// TIA Portal V19 export
FUNCTION_BLOCK "MatLub_FB"   // FB104, LAD
TITLE = MATERIAL LUBRICATION
// stored: MemoryReserve 100, SetENOAutomatically false
   VAR_INPUT
      AreaInterface : "AreaInterface";
      DSI : "udt_DeviceSafetyInterface";
      DataIn : Struct
         Pb_Stop : Bool;
         Pb_Start : Bool;
         SensorLevel : Bool;
      END_STRUCT;
      CoordinationIn : Struct
         MaterialMoving : Bool;
      END_STRUCT;
      Config : Struct
         EnableWngSystemOff : Bool;
         LowTankLevelDly : Time;
      END_STRUCT;
   END_VAR
   VAR_OUTPUT
      MachineInterface : "MachineInterface";
      DataOut : Struct
         SolenoidValve : Bool;
         Lamp : Bool;
      END_STRUCT;
      CoordinationOut : Struct
         IsRunning : Bool;
      END_STRUCT;
   END_VAR
   VAR_IN_OUT
      Parameter : Struct
         SystemOnOff : Bool;
         DelayOff : Time;
      END_STRUCT;
   END_VAR
   VAR
      Sts : Struct
         AlarmsPresence : Bool;
         WarningsPresence : Bool;
         IsStandstill : Bool;
         RunReq : Bool;
         GenCondition { ExternalAccessible := 'False'; ExternalVisible := 'False'; ExternalWritable := 'False'} : Bool;
      END_STRUCT;
      Ctrl : Struct
         RstAlarms : Bool;
         StopDueDoorOpeningRequest : Bool;
         StopSafeStandstill : Bool;
         SafeMotion : Bool;
         StopInPhase : Bool;
         StopProgrammed : Bool;
         StopAborting : Bool;
         ManStart : Bool;
         AutStart : Bool;
      END_STRUCT;
      Alr : Struct
         LowTankLevel : Bool;
      END_STRUCT;
      Wng : Struct
         NoAutReady : Bool;
         SystemOff : Bool;
      END_STRUCT;
      TON_DelayBlowerStop : IEC_TIMER;
      TON_LowTankLevel : IEC_TIMER;
      AckRstAlarms : Bool;
      PbStart_PEAux : Bool;
   END_VAR
   VAR_TEMP   // added for the SCL form of the ladder/FBD networks
      _w1 : Bool;
   END_VAR
BEGIN

REGION Network 1 (SCL): Reset alarms command
   #Ctrl.RstAlarms := #AreaInterface.RstAlarms AND NOT #AckRstAlarms; 
   #AckRstAlarms := #AreaInterface.RstAlarms;

   IF    #Ctrl.RstAlarms THEN
       #Wng.NoAutReady := FALSE;
       #Alr.LowTankLevel := FALSE;
     END_IF;
END_REGION

REGION Network 2: Warning Pump / Blower off
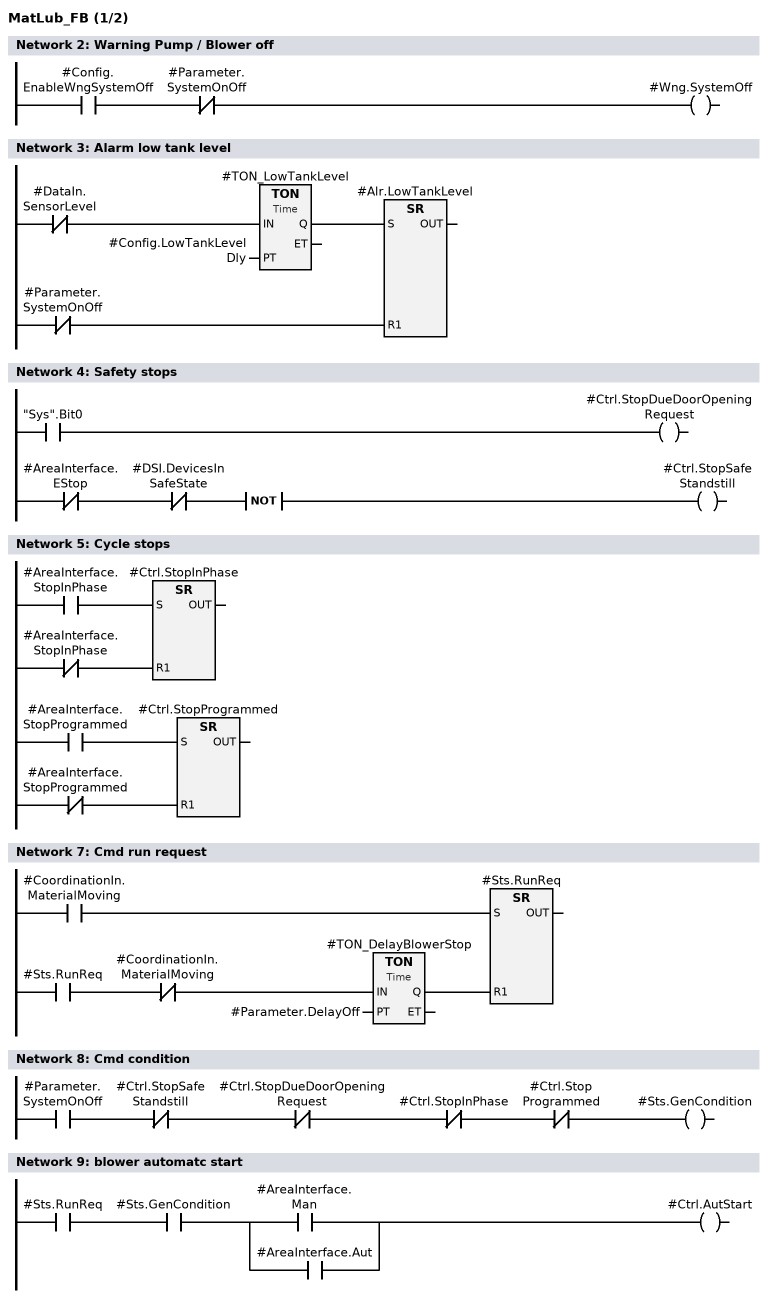
   RUNG wire#powerrail
      Contact( #Config.EnableWngSystemOff )
      I_Contact( #Parameter.SystemOnOff )
      Coil( #Wng.SystemOff )
   END_RUNG
   // the same network as SCL:
   #Wng.SystemOff := #Config.EnableWngSystemOff AND NOT #Parameter.SystemOnOff;
END_REGION

REGION Network 3: Alarm low tank level
   RUNG wire#powerrail
      I_Contact( #DataIn.SensorLevel )
      { S7_Templates := "time_type := Time" } #TON_LowTankLevel.TON(pt := #Config.LowTankLevelDly, et =>)
      S_SR(operand := #Alr.LowTankLevel, r1 := wire#w1)
   END_RUNG
   RUNG wire#powerrail
      I_Contact( #Parameter.SystemOnOff )
   END_RUNG wire#w1
   // the same network as SCL:
   #TON_LowTankLevel.TON(IN := NOT #DataIn.SensorLevel, PT := #Config.LowTankLevelDly);
   IF #TON_LowTankLevel.Q THEN
       #Alr.LowTankLevel := TRUE;   // SR flip-flop
   END_IF;
   IF NOT #Parameter.SystemOnOff THEN #Alr.LowTankLevel := FALSE; END_IF;
END_REGION

REGION Network 4: Safety stops
   RUNG wire#powerrail
      Contact( "Sys".Bit0 )
      Coil( #Ctrl.StopDueDoorOpeningRequest )
   END_RUNG
   RUNG wire#powerrail
      I_Contact( #AreaInterface.EStop )
      I_Contact( #DSI.DevicesInSafeState )
      Not()
      Coil( #Ctrl.StopSafeStandstill )
   END_RUNG
   // the same network as SCL:
   #Ctrl.StopDueDoorOpeningRequest := "Sys".Bit0;
   #Ctrl.StopSafeStandstill := NOT (NOT #AreaInterface.EStop AND NOT #DSI.DevicesInSafeState);
END_REGION

REGION Network 5: Cycle stops
   RUNG wire#powerrail
      Contact( #AreaInterface.StopInPhase )
      S_SR(operand := #Ctrl.StopInPhase, r1 := wire#w1)
   END_RUNG
   RUNG wire#powerrail
      I_Contact( #AreaInterface.StopInPhase )
   END_RUNG wire#w1
   RUNG wire#powerrail
      Contact( #AreaInterface.StopProgrammed )
      S_SR(operand := #Ctrl.StopProgrammed, r1 := wire#w2)
   END_RUNG
   RUNG wire#powerrail
      I_Contact( #AreaInterface.StopProgrammed )
   END_RUNG wire#w2
   // the same network as SCL:
   IF #AreaInterface.StopInPhase THEN
       #Ctrl.StopInPhase := TRUE;   // SR flip-flop
   END_IF;
   IF NOT #AreaInterface.StopInPhase THEN #Ctrl.StopInPhase := FALSE; END_IF;
   IF #AreaInterface.StopProgrammed THEN
       #Ctrl.StopProgrammed := TRUE;   // SR flip-flop
   END_IF;
   IF NOT #AreaInterface.StopProgrammed THEN #Ctrl.StopProgrammed := FALSE; END_IF;
END_REGION

REGION Network 6: <<< BLOWER >>> / <<< COMAMND >>>
END_REGION

REGION Network 7: Cmd run request
   RUNG wire#powerrail
      Contact( #CoordinationIn.MaterialMoving )
      S_SR(operand := #Sts.RunReq, r1 := wire#w1)
   END_RUNG
   RUNG wire#powerrail
      Contact( #Sts.RunReq )
      I_Contact( #CoordinationIn.MaterialMoving )
      { S7_Templates := "time_type := Time" } #TON_DelayBlowerStop.TON(pt := #Parameter.DelayOff, et =>)
   END_RUNG wire#w1
   // the same network as SCL:
   #TON_DelayBlowerStop.TON(IN := #Sts.RunReq AND NOT #CoordinationIn.MaterialMoving, PT := #Parameter.DelayOff);
   IF #CoordinationIn.MaterialMoving THEN
       #Sts.RunReq := TRUE;   // SR flip-flop
   END_IF;
   IF #TON_DelayBlowerStop.Q THEN #Sts.RunReq := FALSE; END_IF;
END_REGION

REGION Network 8: Cmd condition
   RUNG wire#powerrail
      Contact( #Parameter.SystemOnOff )
      I_Contact( #Ctrl.StopSafeStandstill )
      I_Contact( #Ctrl.StopDueDoorOpeningRequest )
      I_Contact( #Ctrl.StopInPhase )
      I_Contact( #Ctrl.StopProgrammed )
      Coil( #Sts.GenCondition )
   END_RUNG
   // the same network as SCL:
   #Sts.GenCondition := #Parameter.SystemOnOff AND NOT #Ctrl.StopSafeStandstill AND NOT #Ctrl.StopDueDoorOpeningRequest AND NOT #Ctrl.StopInPhase AND NOT #Ctrl.StopProgrammed;
END_REGION

REGION Network 9: blower automatc start
   RUNG wire#powerrail
      Contact( #Sts.RunReq )
      Contact( #Sts.GenCondition )
      wire#w1
      Contact( #AreaInterface.Man )
      wire#w2
      Coil( #Ctrl.AutStart )
   END_RUNG
   RUNG wire#w1
      Contact( #AreaInterface.Aut )
   END_RUNG wire#w2
   // the same network as SCL:
   #Ctrl.AutStart := #Sts.RunReq AND #Sts.GenCondition AND (#AreaInterface.Man OR #AreaInterface.Aut);
END_REGION

REGION Network 10: Blower manual start
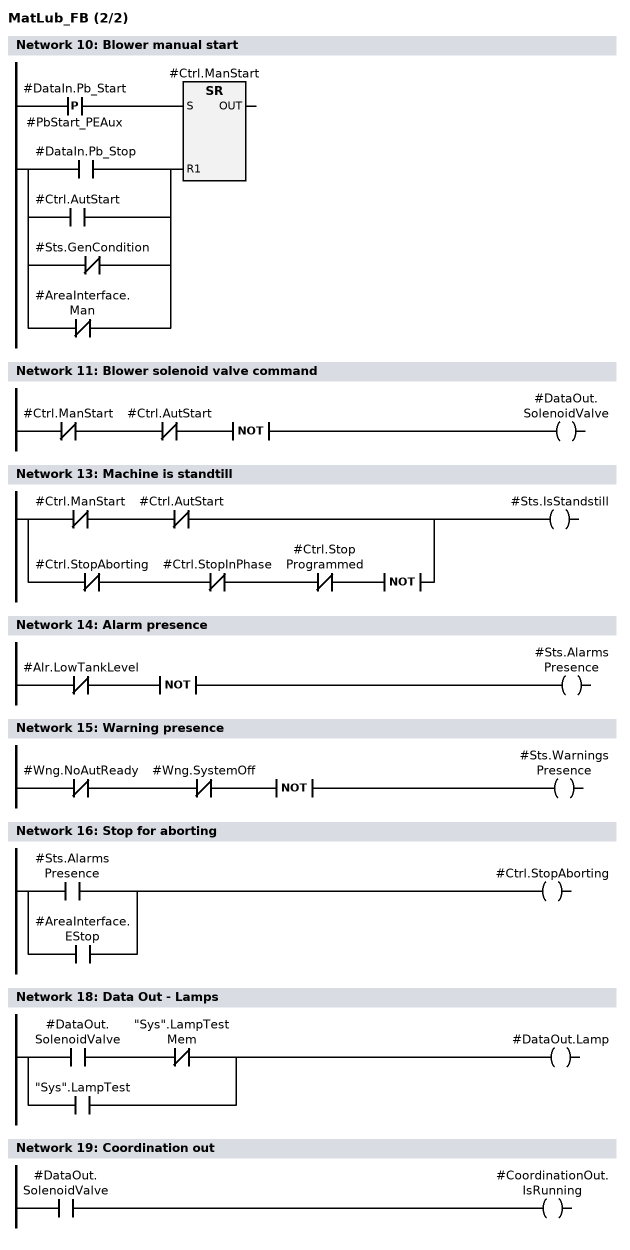
   RUNG wire#powerrail
      P_Contact(operand := #DataIn.Pb_Start, bit := #PbStart_PEAux)
      S_SR(operand := #Ctrl.ManStart, r1 := wire#w1)
   END_RUNG
   RUNG wire#powerrail
      Contact( #DataIn.Pb_Stop )
   END_RUNG wire#w1
   RUNG wire#powerrail
      Contact( #Ctrl.AutStart )
   END_RUNG wire#w1
   RUNG wire#powerrail
      I_Contact( #Sts.GenCondition )
   END_RUNG wire#w1
   RUNG wire#powerrail
      I_Contact( #AreaInterface.Man )
   END_RUNG wire#w1
   // the same network as SCL:
   #_w1 := #DataIn.Pb_Start AND NOT #PbStart_PEAux;   // rising edge of #DataIn.Pb_Start
   #PbStart_PEAux := #DataIn.Pb_Start;
   IF #_w1 THEN
       #Ctrl.ManStart := TRUE;   // SR flip-flop
   END_IF;
   IF #DataIn.Pb_Stop OR #Ctrl.AutStart OR NOT #Sts.GenCondition OR NOT #AreaInterface.Man THEN
       #Ctrl.ManStart := FALSE;
   END_IF;
END_REGION

REGION Network 11: Blower solenoid valve command
   RUNG wire#powerrail
      I_Contact( #Ctrl.ManStart )
      I_Contact( #Ctrl.AutStart )
      Not()
      Coil( #DataOut.SolenoidValve )
   END_RUNG
   // the same network as SCL:
   #DataOut.SolenoidValve := NOT (NOT #Ctrl.ManStart AND NOT #Ctrl.AutStart);
END_REGION

REGION Network 12: <<< >>>
END_REGION

REGION Network 13: Machine is standtill
   RUNG wire#powerrail
      I_Contact( #Ctrl.ManStart )
      I_Contact( #Ctrl.AutStart )
      wire#w1
      Coil( #Sts.IsStandstill )
   END_RUNG
   RUNG wire#powerrail
      I_Contact( #Ctrl.StopAborting )
      I_Contact( #Ctrl.StopInPhase )
      I_Contact( #Ctrl.StopProgrammed )
      Not()
   END_RUNG wire#w1
   // the same network as SCL:
   #Sts.IsStandstill := (NOT #Ctrl.ManStart AND NOT #Ctrl.AutStart) OR NOT (NOT #Ctrl.StopAborting AND NOT #Ctrl.StopInPhase AND NOT #Ctrl.StopProgrammed);
END_REGION

REGION Network 14: Alarm presence
   RUNG wire#powerrail
      I_Contact( #Alr.LowTankLevel )
      Not()
      Coil( #Sts.AlarmsPresence )
   END_RUNG
   // the same network as SCL:
   #Sts.AlarmsPresence := NOT (NOT #Alr.LowTankLevel);
END_REGION

REGION Network 15: Warning presence
   RUNG wire#powerrail
      I_Contact( #Wng.NoAutReady )
      I_Contact( #Wng.SystemOff )
      Not()
      Coil( #Sts.WarningsPresence )
   END_RUNG
   // the same network as SCL:
   #Sts.WarningsPresence := NOT (NOT #Wng.NoAutReady AND NOT #Wng.SystemOff);
END_REGION

REGION Network 16: Stop for aborting
   RUNG wire#powerrail
      Contact( #Sts.AlarmsPresence )
      wire#w1
      Coil( #Ctrl.StopAborting )
   END_RUNG
   RUNG wire#powerrail
      Contact( #AreaInterface.EStop )
   END_RUNG wire#w1
   // the same network as SCL:
   #Ctrl.StopAborting := #Sts.AlarmsPresence OR #AreaInterface.EStop;
END_REGION

REGION Network 17 (SCL): Collect machine to area interface
   // Status machine ready
   #MachineInterface.AutReady := #AreaInterface.Aut AND NOT #Sts.AlarmsPresence;
   // Status machine aborting
   #MachineInterface.Aborting := #Ctrl.StopAborting;
   // Status Ack Stop in phase
   #MachineInterface.AckStopInPhase := #Ctrl.StopInPhase AND #MachineInterface.MotionsStandStill;
   // Status Ack Stop programmed
   #MachineInterface.AckStopProgrammed := #Ctrl.StopProgrammed AND #MachineInterface.MotionsStandStill;
   // Status Motion standtill
   #MachineInterface.MotionsStandStill := #Sts.IsStandstill;
   // Status Alarm presence
   #MachineInterface.AlarmsPresence := #Sts.AlarmsPresence;
   // Status Warning presence
   #MachineInterface.WarningPresence := #Sts.WarningsPresence;

   // Warning machine not automatic ready
   IF #AreaInterface.CheckAutReady AND NOT #MachineInterface.AutReady THEN
     #Wng.NoAutReady := false;
   END_IF;
END_REGION

REGION Network 18: Data Out - Lamps
   RUNG wire#powerrail
      Contact( #DataOut.SolenoidValve )
      I_Contact( "Sys".LampTestMem )
      wire#w1
      Coil( #DataOut.Lamp )
   END_RUNG
   RUNG wire#powerrail
      Contact( "Sys".LampTest )
   END_RUNG wire#w1
   // the same network as SCL:
   #DataOut.Lamp := (#DataOut.SolenoidValve AND NOT "Sys".LampTestMem) OR "Sys".LampTest;
END_REGION

REGION Network 19: Coordination out
   RUNG wire#powerrail
      Contact( #DataOut.SolenoidValve )
      Coil( #CoordinationOut.IsRunning )
   END_RUNG
   // the same network as SCL:
   #CoordinationOut.IsRunning := #DataOut.SolenoidValve;
END_REGION
END_FUNCTION_BLOCK
